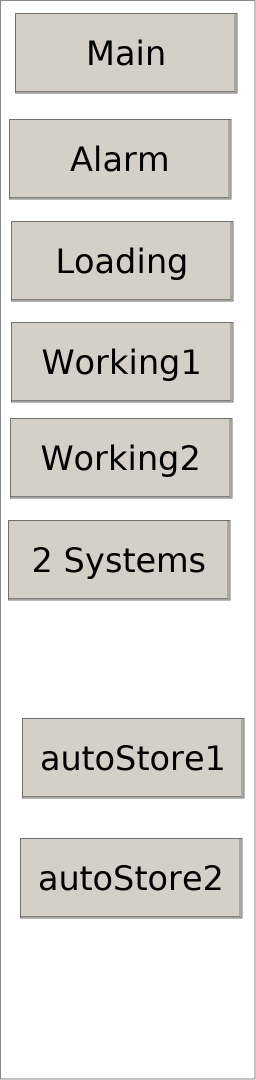
VISUALIZATION Menu  // 256x1080
    Button (9,119 222x80), "Alarm", colour toggle: G_HMI.iMainFrame =1
        p573394764: 16#FF000000 OR ( 16#FF00FF00)
        OnMouseDown: execute { G_HMI.iMainFrame	:= 1; }
    Button (15,13 222x80), "Main", colour toggle: G_HMI.iMainFrame =0
        p573394764: 16#FF000000 OR ( 16#FF00FF00)
        OnMouseDown: execute { G_HMI.iMainFrame	:= 0; }
    Button (11,221 222x80), "Loading", colour toggle: G_HMI.iMainFrame =2
        p573394764: 16#FF000000 OR ( 16#FF00FF00)
        OnMouseDown: execute { G_HMI.iMainFrame	:= 2; }
    Button (11,322 222x80), "Working1", colour toggle: G_HMI.iMainFrame =3
        p573394764: 16#FF000000 OR ( 16#FF00FF00)
        OnMouseDown: execute { G_HMI.iMainFrame	:= 3; }
    Button (10,418 222x80), "Working2", colour toggle: G_HMI.iMainFrame =4
        p573394764: 16#FF000000 OR ( 16#FF00FF00)
        OnMouseDown: execute { G_HMI.iMainFrame	:= 4; }
    Button (8,520 222x80), "2 Systems", colour toggle: G_HMI.iMainFrame =5
        p573394764: 16#FF000000 OR ( 16#FF00FF00)
        OnMouseDown: execute { G_HMI.iMainFrame	:= 5; }
    Button (22,718 222x80), "autoStore1", colour toggle: G_HMI.iMainFrame =6
        p573394764: 16#FF000000 OR ( 16#FF00FF00)
        OnMouseDown: execute { G_HMI.iMainFrame	:= 6; }
    Button (20,838 222x80), "autoStore2", colour toggle: G_HMI.iMainFrame =7
        p573394764: 16#FF000000 OR ( 16#FF00FF00)
        OnMouseDown: execute { G_HMI.iMainFrame	:= 7; }
END_VISUALIZATION

(* stored: Version 1.1.0.1, ProductVersion 3.1.4024.12
   Visu Menu: Id {2c1cc129-5e67-4f8a-b890-3aee9edbaf72} *)
